// TIA Portal V20 export
DATA_BLOCK "RealDbName"   // DB7
   VAR
      IO { S7_SetPoint := 'True'} : "TypeDOL";
   END_VAR
BEGIN
END_DATA_BLOCK
